TYPE ST_RegParams : 
STRUCT
	fCtrlCycleTime	 : LREAL;
	fKp		 : LREAL;
	fTn		 : LREAL;
	fTv		 : LREAL;
	fTd		 : LREAL;
END_STRUCT
END_TYPE

(* stored: Version 1.1.0.1, ProductVersion 3.1.4024.11
   DUT ST_RegParams: Id {f11cdf90-dd6b-4074-bb3b-722a4877c1f5} *)
